(* CODESYS project TestSuite_V1.1.3.library
   Author: Simmel Florian
   Version: 1.1.3
   Title: Tc3_PlcTestSuite
   DefaultNamespace: Tc3_PlcTestSuite
   Placeholder: Tc3_PlcTestSuite
   Company: Simmel

Project tree, tasks and I/O mapping:
  libraries: Tc2_EtherCAT, * (Beckhoff Automation GmbH); Tc2_Standard, * (Beckhoff Automation GmbH); Tc2_System, * (Beckhoff Automation GmbH); Tc2_Utilities, * (Beckhoff Automation GmbH); Tc3_EventLogger, * (Beckhoff Automation GmbH); Tc3_JsonXml, * (Beckhoff Automation GmbH)
  Functions/
    function block AdsLogger [ST]: FB_Init, LogMessage
    function GetValueString [ST]
    function block JUnitResultFile [ST]: AddTestCaseResult, AddTestSuite, AddTestSuiteStatistics, Cyclic, FB_Init, FindSuiteNode, Initialize, Initialized, Path, SaveResult, SuiteOverflowCount
    function block Stopwatch [ST]: Elapsed, Lap, Running, Start, Stop
  Interfaces/
    interface I_TestOperation: AssertEqual, Duration, ExecuteTest, State, TestId, TestSuiteName
    interface I_TestSuite: Duration, ReRunIndividualTest, ReRunTests, Test
    interface I_UnitTestResultFile: AddTestCaseResult, AddTestSuite, AddTestSuiteStatistics, Cyclic, Initialize, Initialized, Path, SaveResult
  Project Information/
    function F_GetCompany [ST]
    function F_GetTitle [ST]
    function F_GetVersion [ST]
  Structures/
    data type E_TestStatus
    data type ST_TestDefinition
  Version/
    global variables Global_Version
  global variables GlobalTestSuite
  function block Test [ST]: AssertEqual, Duration, ExecuteTest, ReportAssert, ResultFileFunction, State, TestId, TestSuiteName
  function block TestSuite [ST]: Duration, FB_Init, ReRunIndividualTest, ReRunTests, ResultFileFunction, Test, TestOverflowCount, TestSuiteName
  global variables TestSuiteParameter
*)

// Structures/E_TestStatus
{attribute 'qualified_only'}
{attribute 'strict'}
{attribute 'to_string'}
TYPE E_TestStatus : (
		Init := 0,
		Running,
		DoneOk,
		DoneFailed
	);
END_TYPE

// Structures/ST_TestDefinition
TYPE ST_TestDefinition :
	STRUCT
		TestId : T_MaxString;
		Status : E_TestStatus;
	END_STRUCT
END_TYPE

// Version/Global_Version
{attribute 'TcGenerated'}
{attribute 'no-analysis'}
{attribute 'linkalways'}
// This function has been automatically generated from the project information.
VAR_GLOBAL CONSTANT
	{attribute 'const_non_replaced'}
	stLibVersion_Tc3_PlcTestSuite : ST_LibVersion := (iMajor := 1, iMinor := 1, iBuild := 3, iRevision := 0, nFlags := 0, sVersion := '1.1.3');
END_VAR

// GlobalTestSuite
VAR_GLOBAL
	JUnitResultFile   : JUnitResultFile<TestSuiteParameter.MaxTestSuiteCount>(TestSuiteParameter.DefaultPath);
	TestSuite		  : TestSuite<TestSuiteParameter.MaxTestCount>(ResultFile := JUnitResultFile);
	AdsLoggingEnabled : BOOL := FALSE;
END_VAR

// TestSuiteParameter
{attribute 'qualified_only'}
VAR_GLOBAL CONSTANT
	MaxTestCount	  : DINT   := 50;
	MaxTestSuiteCount : DINT   := 10;
	DefaultPath		  : STRING := 'C:\ProgramData\Beckhoff\TwinCAT\3.1\Boot\TEST_Result.xml';
END_VAR

// Functions/AdsLogger
FUNCTION_BLOCK AdsLogger
VAR
    Enabled : REFERENCE TO  BOOL;
END_VAR

//FB_Init is always available implicitly and it is used primarily for initialization.
//The return value is not evaluated. For a specific influence, you can also declare the
//methods explicitly and provide additional code there with the standard initialization
//code. You can evaluate the return value.
METHOD FB_Init: BOOL
VAR_INPUT
    bInitRetains: BOOL; // TRUE: the retain variables are initialized (reset warm / reset cold)
    bInCopyCode: BOOL;  // TRUE: the instance will be copied to the copy code afterward (online change) 
    Enabled : REFERENCE TO BOOL;  
END_VAR
THIS^.Enabled Ref= Enabled;
END_METHOD

METHOD LogMessage
VAR_INPUT
	Message : STRING;
END_VAR
IF THIS^.Enabled THEN
	ADSLOGSTR(ADSLOG_MSGTYPE_HINT, Message, '');
END_IF
END_METHOD

END_FUNCTION_BLOCK

// Functions/GetValueString
FUNCTION GetValueString : STRING
VAR_INPUT
	Symbol : ANY;
END_VAR

VAR
	ubuff  : ULINT;
	sibuff : SINT;
	ibuff  : INT;
	dibuff : DINT;
	libuff : LINT;
	rbuff  : REAL;
    lrbuff : LREAL;
	sbuff  : STRING(255);
	wsbuff : WSTRING(255);
	x	   : INT; // loop var for STRING and WSTRING
END_VAR

GetValueString := '';
CASE Symbol.TypeClass OF
	__SYSTEM.TYPE_CLASS.TYPE_BOOL:
		memcpy(ADR(ubuff), Symbol.pValue, TO_UDINT(Symbol.diSize));
		GetValueString := TO_STRING(TO_BOOL(TO_LREAL(ubuff)));

	__SYSTEM.TYPE_CLASS.TYPE_BYTE, __SYSTEM.TYPE_CLASS.TYPE_USINT, __SYSTEM.TYPE_CLASS.TYPE_WORD, __SYSTEM.TYPE_CLASS.TYPE_UINT, __SYSTEM.TYPE_CLASS.TYPE_DWORD, __SYSTEM.TYPE_CLASS.TYPE_UDINT, __SYSTEM.TYPE_CLASS.TYPE_LWORD, __SYSTEM.TYPE_CLASS.TYPE_ULINT:
		memcpy(ADR(ubuff), Symbol.pValue, TO_UDINT(Symbol.diSize));
		GetValueString := LREAL_TO_FMTSTR(TO_LREAL(ubuff), 0, FALSE);

	__SYSTEM.TYPE_CLASS.TYPE_SINT:
		memcpy(ADR(sibuff), Symbol.pValue, TO_UDINT(Symbol.diSize));
		GetValueString := LREAL_TO_FMTSTR(TO_LREAL(sibuff), 0, FALSE);

	__SYSTEM.TYPE_CLASS.TYPE_INT:
		memcpy(ADR(ibuff), Symbol.pValue, TO_UDINT(Symbol.diSize));
		GetValueString := LREAL_TO_FMTSTR(TO_LREAL(ibuff), 0, FALSE);

	__SYSTEM.TYPE_CLASS.TYPE_DINT:
		memcpy(ADR(dibuff), Symbol.pValue, TO_UDINT(Symbol.diSize));
		GetValueString := LREAL_TO_FMTSTR(TO_LREAL(dibuff), 0, FALSE);

	__SYSTEM.TYPE_CLASS.TYPE_LINT:
		memcpy(ADR(libuff), Symbol.pValue, TO_UDINT(Symbol.diSize));
		GetValueString := LREAL_TO_FMTSTR(TO_LREAL(libuff), 0, FALSE);

	__SYSTEM.TYPE_CLASS.TYPE_REAL, __SYSTEM.TYPE_CLASS.TYPE_LREAL:
		IF Symbol.TypeClass = __SYSTEM.TYPE_CLASS.TYPE_REAL THEN
			memcpy(ADR(rbuff), Symbol.pValue, TO_UDINT(Symbol.diSize));
			GetValueString := LREAL_TO_FMTSTR(TO_LREAL(rbuff), 5, TRUE);
		ELSIF Symbol.TypeClass = __SYSTEM.TYPE_CLASS.TYPE_LREAL THEN
			memcpy(ADR(lrbuff), Symbol.pValue, TO_UDINT(Symbol.diSize));
			GetValueString := LREAL_TO_FMTSTR(TO_LREAL(lrbuff), 5, TRUE);
		END_IF

	__SYSTEM.TYPE_CLASS.TYPE_STRING, __SYSTEM.TYPE_CLASS.TYPE_WSTRING:
		IF Symbol.TypeClass = __SYSTEM.TYPE_CLASS.TYPE_STRING THEN
			MEMCPY(ADR(sbuff), Symbol.pValue, MIN(SIZEOF(sbuff), TO_UDINT(Symbol.diSize)));
		ELSIF Symbol.TypeClass = __SYSTEM.TYPE_CLASS.TYPE_WSTRING THEN
			MEMCPY(ADR(wsbuff), Symbol.pValue, MIN(SIZEOF(wsbuff), TO_UDINT(Symbol.diSize)));
			WSTRING_TO_STRING2(ADR(sbuff), ADR(wsbuff), SIZEOF(sbuff));
		END_IF

		GetValueString := sbuff;
END_CASE

END_FUNCTION

// Functions/JUnitResultFile
FUNCTION_BLOCK JUnitResultFile
VAR_GENERIC CONSTANT
	_MaxTestSuiteCount : DINT := 10;
END_VAR IMPLEMENTS I_UnitTestResultFile
VAR
	_Initialized, Write										   : BOOL;
	XmlDomParser											   : FB_XmlDomParser;
	RootNode, TestSuitesNode, TestSuite, TestCase, TestCaseSub : SXmlNode;
	_Path													   : STRING;
	SuiteNames												   : ARRAY[0.._MaxTestSuiteCount] OF STRING;
	SuiteNodes												   : ARRAY[0.._MaxTestSuiteCount] OF SXmlNode;
	SuiteCount												   : DINT;
	DoneMessage												   : FB_TcMessage;
	Source													   : FB_TcSourceInfo;
	_SuiteOverflowCount										   : UDINT;
END_VAR

METHOD AddTestCaseResult
VAR_INPUT
	TestClassName	: STRING;
	TestName		: STRING;
	Duration		: LREAL;
	FailtureMessage : STRING := '';
	FailtureType	: STRING := '';
	FailtureNote	: STRING := '';
END_VAR
VAR
	SuiteNode : SXmlNode;
END_VAR
IF NOT Initialized THEN
	RETURN;
END_IF

SuiteNode := FindSuiteNode(TestClassName);
IF SuiteNode = 0 THEN
	RETURN;
END_IF

TestCase := XmlDomParser.AppendChild(SuiteNode,
									 'testcase',
									 '',
									 FALSE);

XmlDomParser.AppendAttribute(TestCase, 'classname', TestClassName);
XmlDomParser.AppendAttribute(TestCase, 'name', TestName);
XmlDomParser.AppendAttributeAsDouble(TestCase, 'time', Duration);
IF FailtureType <> '' THEN
	TestCaseSub := XmlDomParser.AppendChild(TestCase,
											'failure',
											FailtureNote,
											FALSE);

	XmlDomParser.AppendAttribute(TestCaseSub, 'message', FailtureMessage);
	XmlDomParser.AppendAttribute(TestCaseSub, 'type', FailtureType);
END_IF
END_METHOD

METHOD AddTestSuite
VAR_INPUT
	Name : STRING;
END_VAR
VAR
	ResultString : T_MaxString;
END_VAR
IF NOT Initialized THEN
	RETURN;
END_IF

// Reuse the existing node if this suite name was already added (shared result file across multiple TestSuite instances)
TestSuite := FindSuiteNode(Name);
IF TestSuite <> 0 THEN
	RETURN;
END_IF

TestSuite := XmlDomParser.AppendChild(TestSuitesNode,
									  'testsuite',
									  '',
									  FALSE);

XmlDomParser.AppendAttribute(TestSuite, 'name', name);

IF SuiteCount <= _MaxTestSuiteCount THEN
	SuiteNames[SuiteCount] := Name;
	SuiteNodes[SuiteCount] := TestSuite;
	SuiteCount			   := SuiteCount + 1;
ELSE
	_SuiteOverflowCount := _SuiteOverflowCount + 1;

	Source.sName := Name;
	DoneMessage.Create(eventClass	:= TC_EVENT_CLASSES.TestEvents,
					   nEventId		:= 1,
					   eSeverity	:= TcEventSeverity.Error,
					   ipSourceInfo := Source);

	ResultString := CONCAT('TestSuite not added, max TestSuites exeeded - ', TO_STRING(_MaxTestSuiteCount));
	DoneMessage.ipArguments.AddString(ResultString);
	DoneMessage.Send(0);
	Source.Clear();
	DoneMessage.Release();
END_IF
END_METHOD

METHOD AddTestSuiteStatistics
VAR_INPUT
	Name	  : STRING;
	Tests	  : UDINT;
	Failtures : UDINT := 0;
	Errors	  : UDINT := 0;
	Skipped	  : UDINT := 0;
	Duration  : LREAL;
END_VAR
VAR
	SuiteNode : SXmlNode;
END_VAR
IF NOT Initialized THEN
	RETURN;
END_IF

SuiteNode := FindSuiteNode(Name);
IF SuiteNode = 0 THEN
	RETURN;
END_IF

XmlDomParser.AppendAttributeAsUint(SuiteNode, 'tests', Tests);
XmlDomParser.AppendAttributeAsUint(SuiteNode, 'failtures', Failtures);
XmlDomParser.AppendAttributeAsUint(SuiteNode, 'errors', Errors);
XmlDomParser.AppendAttributeAsUint(SuiteNode, 'skipped', Skipped);
XmlDomParser.AppendAttributeAsDouble(SuiteNode, 'time', Duration);
END_METHOD

METHOD Cyclic
XmlDomParser.SaveDocumentToFile(_Path, Write);
END_METHOD

//FB_Init is always available implicitly and it is used primarily for initialization.

//The return value is not evaluated. For a specific influence, you can also declare the

//methods explicitly and provide additional code there with the standard initialization

//code. You can evaluate the return value.
METHOD FB_Init : BOOL
VAR_INPUT
	bInitRetains : BOOL; // TRUE: the retain variables are initialized (reset warm / reset cold)
	bInCopyCode	 : BOOL; // TRUE: the instance will be copied to the copy code afterward (online change)
	Path		 : STRING;
END_VAR
_Path := Path;
END_METHOD

METHOD PRIVATE FindSuiteNode : SXmlNode
VAR_INPUT
	Name : STRING;
END_VAR
VAR
	i : DINT;
END_VAR
FindSuiteNode := 0;

FOR i := 0 TO SuiteCount - 1 DO
	IF SuiteNames[i] = Name THEN
		FindSuiteNode := SuiteNodes[i];
		RETURN;
	END_IF
END_FOR
END_METHOD

METHOD Initialize
VAR_INPUT
	ReInitialize : BOOL := FALSE;
END_VAR
IF Initialized AND NOT ReInitialize THEN
	RETURN;
END_IF

XmlDomParser.NewDocument();
RootNode	   := XmlDomParser.GetDocumentNode();
TestSuitesNode := XmlDomParser.AppendChild(RootNode,
										   'testsuites',
										   '',
										   FALSE);

SuiteCount	 := 0;
_Initialized := TRUE;
END_METHOD

{attribute 'monitoring' := 'call'}
PROPERTY Initialized : BOOL
GET
Initialized := _Initialized;
END_GET
END_PROPERTY

{attribute 'monitoring' := 'call'}
PROPERTY Path : STRING
SET
_Path := Path;
END_SET
END_PROPERTY

METHOD SaveResult
IF NOT Initialized THEN
	RETURN;
END_IF

Write := TRUE;
END_METHOD

{attribute 'monitoring' := 'call'}
PROPERTY SuiteOverflowCount : UDINT
GET
SuiteOverflowCount := _SuiteOverflowCount;
END_GET
END_PROPERTY

END_FUNCTION_BLOCK

// Interfaces/I_UnitTestResultFile
INTERFACE I_UnitTestResultFile EXTENDS __SYSTEM.IQueryInterface

METHOD AddTestCaseResult
VAR_INPUT
	TestClassName	: STRING;
	TestName		: STRING;
	Duration		: LREAL;
	FailtureMessage : STRING := '';
	FailtureType	: STRING := '';
	FailtureNote	: STRING := '';
END_VAR
END_METHOD

METHOD AddTestSuite
VAR_INPUT
	Name	  : STRING;
END_VAR
END_METHOD

METHOD AddTestSuiteStatistics
VAR_INPUT
	Name	  : STRING;
	Tests	  : UDINT;
	Failtures : UDINT := 0;
	Errors	  : UDINT := 0;
	Skipped	  : UDINT := 0;
	Duration  : LREAL;
END_VAR
END_METHOD

METHOD Cyclic
VAR_INPUT
END_VAR
END_METHOD

METHOD Initialize
VAR_INPUT
	ReInitialize : BOOL := FALSE;
END_VAR
END_METHOD

{attribute 'monitoring' := 'call'}
PROPERTY Initialized : BOOL
GET
END_GET
END_PROPERTY

{attribute 'monitoring' := 'call'}
PROPERTY Path : STRING
SET
END_SET
END_PROPERTY

METHOD SaveResult
VAR_INPUT
END_VAR
END_METHOD

END_INTERFACE

// TestSuite
FUNCTION_BLOCK TestSuite
VAR_GENERIC CONSTANT
	_MaxTestCount : DINT := 10;
END_VAR IMPLEMENTS I_TestSuite
VAR
	_TestSuiteName	  : STRING;
	TestCollection	  : ARRAY[0.._MaxTestCount] OF Test;
	NoAction		  : Test := (TestId := 'No Action', State := E_TestStatus.DoneOk);
	ActiveTest		  : DINT;
	DoneMessage		  : FB_TcMessage;
	Source			  : FB_TcSourceInfo;
	TotalTestCount	  : UDINT := 0;
	TotalOkTestCount  : UDINT := 0;
	TotalNokTestCount : UDINT := 0;
	Complete		  : BOOL;
	ResultFile		  : I_UnitTestResultFile;
	_ResultFileAdded  : BOOL;
	CurrentCycle	  : UDINT;
	Stopwatch		  : Stopwatch;
	_TestOverflowCount : UDINT;
END_VAR

{attribute 'monitoring' := 'call'}
PROPERTY Duration : LREAL
GET
Duration := Stopwatch.Elapsed;
END_GET
END_PROPERTY

//FB_Init is always available implicitly and it is used primarily for initialization.

//The return value is not evaluated. For a specific influence, you can also declare the

//methods explicitly and provide additional code there with the standard initialization

//code. You can evaluate the return value.
METHOD FB_Init : BOOL
VAR_INPUT
	bInitRetains : BOOL; // TRUE: the retain variables are initialized (reset warm / reset cold)
	bInCopyCode	 : BOOL; // TRUE: the instance will be copied to the copy code afterward (online change)
	ResultFile	 : I_UnitTestResultFile;
END_VAR
IF ResultFile <> 0 THEN
	THIS^.ResultFile := ResultFile;
END_IF
END_METHOD

{attribute 'TcRpcEnable':='1'}
METHOD ReRunIndividualTest
VAR_INPUT
	TestId : T_MaxString;
END_VAR

VAR
	i : DINT;
END_VAR
FOR i := 0 TO _MaxTestCount DO
	IF TestCollection[i].TestId = TestId THEN
		TestCollection[i].State := E_TestStatus.Init;
		ActiveTest := i;
		Complete := FALSE;
		EXIT;
	END_IF
END_FOR
END_METHOD

{attribute 'TcRpcEnable':='1'}
METHOD ReRunTests
VAR
	i : DINT;
END_VAR
FOR i := 0 TO TestSuiteParameter.MaxTestCount DO
	TestCollection[i].State := E_TestStatus.Init;
	ActiveTest				:= 0;
	Complete				:= FALSE;
	ResultFile.Initialize();
	Stopwatch.Start();
	ResultFile.AddTestSuite(Name := _TestSuiteName);
END_FOR
END_METHOD

PROPERTY ResultFileFunction : I_UnitTestResultFile
SET
ResultFile := ResultFileFunction;
END_SET
END_PROPERTY

METHOD Test : I_TestOperation
VAR_INPUT
	TestId : T_MaxString;
END_VAR

VAR
	ResultString : T_MaxString;
	i			 : DINT;
END_VAR
IF _TestSuiteName = '' THEN
	_TestSuiteName := __POUNAME();
END_IF

IF NOT _ResultFileAdded THEN
	_ResultFileAdded := TRUE;
	ResultFile.Initialize();
	Stopwatch.Start();
	ResultFile.AddTestSuite(Name := _TestSuiteName);
END_IF

IF TwinCAT_SystemInfoVarList._TaskInfo[GETCURTASKINDEXEX()].CycleCount <> CurrentCycle THEN
	CurrentCycle := TwinCAT_SystemInfoVarList._TaskInfo[GETCURTASKINDEXEX()].CycleCount;
	ResultFile.Cyclic();
END_IF

IF NOT Complete THEN
	FOR i := 0 TO _MaxTestCount DO
		TestCollection[i].TestSuiteName		 := _TestSuiteName;
		TestCollection[i].ResultFileFunction := ResultFile;
		// Detect first running test
		IF TestCollection[i].State = E_TestStatus.Running THEN
			ActiveTest := i;
		END_IF

		IF TestCollection[ActiveTest].State >= E_TestStatus.DoneOk THEN
			ActiveTest := 0;
		END_IF

		// Get existing Test
		IF (TestCollection[i].TestId = TestId) THEN
			IF (ActiveTest = i) OR (ActiveTest = 0) THEN
				Test := TestCollection[i];
			ELSE
				Test := NoAction;
			END_IF

			EXIT;
		END_IF

		// Add Test
		IF TestCollection[i].TestId = '' THEN
			TestCollection[i].TestId := TestId;
			Test					 := NoAction;
			EXIT;
		END_IF

		// Out of tests
		IF i = _MaxTestCount THEN
			Test			   := NoAction;
			_TestOverflowCount := _TestOverflowCount + 1;
			Source.sName	   := _TestSuiteName;
			DoneMessage.Create(eventClass	:= TC_EVENT_CLASSES.TestEvents,
							   nEventId		:= 1,
							   eSeverity	:= TcEventSeverity.Error,
							   ipSourceInfo := Source);

			ResultString := CONCAT('Test not added, max Tests exeeded - ', TO_STRING(_MaxTestCount));
			DoneMessage.ipArguments.AddString(ResultString);
			DoneMessage.Send(0);
			Source.Clear();
			DoneMessage.Release();
			Complete := TRUE;
		END_IF
	END_FOR

	// Run Statistic
	TotalTestCount	  := 0;
	TotalOkTestCount  := 0;
	TotalNokTestCount := 0;
	FOR i := 0 TO _MaxTestCount DO
		IF TestCollection[i].TestId <> '' THEN
			TotalTestCount := TotalTestCount + 1;
			IF TestCollection[i].State = E_TestStatus.DoneOk THEN
				TotalOkTestCount := TotalOkTestCount + 1;
			END_IF

			IF TestCollection[i].State = E_TestStatus.DoneFailed THEN
				TotalNokTestCount := TotalNokTestCount + 1;
			END_IF
		END_IF
	END_FOR

	// Tests finished
	IF (TotalTestCount = (TotalOkTestCount + TotalNokTestCount)) AND NOT Complete THEN
		Source.sName := _TestSuiteName;
		DoneMessage.Create(eventClass	:= TC_EVENT_CLASSES.TestEvents,
						   nEventId		:= 1,
						   eSeverity	:= TcEventSeverity.Error,
						   ipSourceInfo := Source);

		ResultString := CONCAT('Completed - ', CONCAT('Total Tests - ', TO_STRING(TotalTestCount)));
		ResultString := CONCAT(ResultString, CONCAT(', OK Tests - ', TO_STRING(TotalOkTestCount)));
		ResultString := CONCAT(ResultString, CONCAT(', Failed Tests - ', TO_STRING(TotalNokTestCount)));
		DoneMessage.ipArguments.AddString(ResultString);
		DoneMessage.Send(0);
		Source.Clear();
		DoneMessage.Release();

		//
		Stopwatch.Stop();
		ResultFile.AddTestSuiteStatistics(Name := _TestSuiteName, Tests := TotalTestCount, Failtures := TotalNokTestCount, Duration := Stopwatch.Elapsed);
		ResultFile.SaveResult();

		//
		Complete := TRUE;
	END_IF
ELSE
	Test := NoAction;
END_IF
END_METHOD

{attribute 'monitoring' := 'call'}
PROPERTY TestOverflowCount : UDINT
GET
TestOverflowCount := _TestOverflowCount;
END_GET
END_PROPERTY

{attribute 'monitoring' := 'call'}
PROPERTY TestSuiteName : STRING
SET
_TestSuiteName := TestSuiteName;
END_SET
END_PROPERTY

END_FUNCTION_BLOCK

// Interfaces/I_TestSuite
INTERFACE I_TestSuite EXTENDS __SYSTEM.IQueryInterface

{attribute 'monitoring' := 'call'}
PROPERTY Duration : LREAL
GET
END_GET
END_PROPERTY

METHOD ReRunIndividualTest
VAR_INPUT
	TestId : T_MaxString;
END_VAR
END_METHOD

METHOD ReRunTests
VAR_INPUT
END_VAR
END_METHOD

METHOD Test : I_TestOperation
VAR_INPUT
	TestId : T_MaxString;
END_VAR
END_METHOD

END_INTERFACE

// Test
FUNCTION_BLOCK Test IMPLEMENTS I_TestOperation
VAR
	_TestSuiteName : STRING;
	_TestId		   : T_MaxString;
	_State		   : E_TestStatus;
	TestMessage	   : FB_TcMessage;
	Source		   : FB_TcSourceInfo;
	Stopwatch	   : Stopwatch;
	ResultFile	   : I_UnitTestResultFile;
	AdsLogger	   : AdsLogger(GlobalTestSuite.AdsLoggingEnabled);
END_VAR

METHOD AssertEqual
VAR_INPUT
	Expected : ANY;
	Actual	 : ANY;
	Epsilon	 : LREAL := 0.000001;
END_VAR

VAR
	nCount		   : DINT;
	StringExpected : T_MaxString;
	StringActual   : T_MaxString;
	LrealExpected  : LREAL;
	LrealActual	   : LREAL;
	RealExpected   : REAL;
	RealActual	   : REAL;
END_VAR
Stopwatch.Stop();
IF Expected.typeclass <> Actual.typeclass THEN
	State := E_TestStatus.DoneFailed;
	ReportAssert('Type missmatch!');
	RETURN;
END_IF

IF Expected.diSize <> Actual.diSize THEN
	State := E_TestStatus.DoneFailed;
	ReportAssert('Type size missmatch!');
	RETURN;
END_IF

// String
IF Expected.TypeClass = __SYSTEM.TYPE_CLASS.TYPE_ANYSTRING OR Expected.TypeClass = __SYSTEM.TYPE_CLASS.TYPE_STRING OR Expected.TypeClass = __SYSTEM.TYPE_CLASS.TYPE_WSTRING OR Expected.TypeClass = __SYSTEM.TYPE_CLASS.TYPE_XSTRING THEN
	MEMCPY(destAddr := ADR(StringExpected), srcAddr := Expected.pValue, n := DINT_TO_UDINT(Expected.diSize));
	MEMCPY(destAddr := ADR(StringActual), srcAddr := Actual.pValue, n := DINT_TO_UDINT(Actual.diSize));
	IF StringExpected <> StringActual THEN
		State := E_TestStatus.DoneFailed;
		ReportAssert(CONCAT(CONCAT('Expected: ', GetValueString(Expected)), CONCAT(' , Actual: ', GetValueString(Actual))));
		RETURN;
	END_IF
ELSIF Expected.TypeClass = __SYSTEM.TYPE_CLASS.TYPE_LREAL THEN
	MEMCPY(destAddr := ADR(LrealExpected), srcAddr := Expected.pValue, n := DINT_TO_UDINT(Expected.diSize));
	MEMCPY(destAddr := ADR(LrealActual), srcAddr := Actual.pValue, n := DINT_TO_UDINT(Actual.diSize));
	IF ((LrealExpected - Epsilon) > LrealActual) OR ((LrealExpected + Epsilon) < LrealActual) THEN
		State := E_TestStatus.DoneFailed;
		ReportAssert(CONCAT(CONCAT('Expected: ', GetValueString(Expected)), CONCAT(' , Actual: ', GetValueString(Actual))));
		RETURN;
	END_IF
ELSIF Expected.TypeClass = __SYSTEM.TYPE_CLASS.TYPE_ANYREAL OR Expected.TypeClass = __SYSTEM.TYPE_CLASS.TYPE_REAL THEN
	MEMCPY(destAddr := ADR(RealExpected), srcAddr := Expected.pValue, n := DINT_TO_UDINT(Expected.diSize));
	MEMCPY(destAddr := ADR(RealActual), srcAddr := Actual.pValue, n := DINT_TO_UDINT(Actual.diSize));
	IF ((RealExpected - Epsilon) > RealActual) OR ((RealExpected + Epsilon) < RealActual) THEN
		State := E_TestStatus.DoneFailed;
		ReportAssert(CONCAT(CONCAT('Expected: ', GetValueString(Expected)), CONCAT(' , Actual: ', GetValueString(Actual))));
		RETURN;
	END_IF
ELSE
	// Byte comparison
	FOR nCount := 0 TO Actual.diSize - 1 DO
		IF Expected.pvalue[nCount] <> Actual.pvalue[nCount] THEN
			State := E_TestStatus.DoneFailed;
			ReportAssert(CONCAT(CONCAT('Expected: ', GetValueString(Expected)), CONCAT(' , Actual: ', GetValueString(Actual))));
			RETURN;
		END_IF
	END_FOR
END_IF

IF ResultFile <> 0 THEN
	ResultFile.AddTestCaseResult(_TestSuiteName, TestId, Stopwatch.Elapsed);
END_IF

AdsLogger.LogMessage(Concat('Test Executed: ', TestId));
State := E_TestStatus.DoneOk;
END_METHOD

{attribute 'monitoring' := 'call'}
PROPERTY Duration : LREAL
GET
Duration := Stopwatch.Elapsed;
END_GET
END_PROPERTY

METHOD ExecuteTest : BOOL
VAR_INPUT
END_VAR
IF State = E_TestStatus.Init THEN
	Stopwatch.Start();
	State := E_TestStatus.Running;
END_IF

ExecuteTest := State = E_TestStatus.Running;
END_METHOD

METHOD PRIVATE ReportAssert
VAR_INPUT
	Reason : STRING := '';
END_VAR

VAR
	ResultString : T_MaxString;
END_VAR
Source.sName := _TestSuiteName;
TestMessage.Create(eventClass	:= TC_EVENT_CLASSES.TestEvents,
				   nEventId		:= 1,
				   eSeverity	:= TcEventSeverity.Error,
				   ipSourceInfo := Source);

ResultString := CONCAT('Test failed - ', TestId);
ResultString := CONCAT(ResultString, '! ');
ResultString := CONCAT(ResultString, Reason);
TestMessage.ipArguments.AddString(ResultString);
TestMessage.Send(0);
Source.Clear();
TestMessage.Release();
AdsLogger.LogMessage(Concat('Test Executed: ', TestId));
IF ResultFile <> 0 THEN
	ResultFile.AddTestCaseResult(_TestSuiteName,
								 TestId,
								 Stopwatch.Elapsed,
								 'Test failed!',
								 'AssertionError',
								 Reason);
END_IF
END_METHOD

PROPERTY ResultFileFunction : I_UnitTestResultFile
SET
ResultFile := ResultFileFunction;
END_SET
END_PROPERTY

{attribute 'monitoring' := 'call'}
PROPERTY State :  E_TestStatus
GET
State := _State;
END_GET
SET
_State := State;
END_SET
END_PROPERTY

{attribute 'monitoring' := 'call'}
PROPERTY TestId : T_MaxString
GET
TestId := _TestId;
END_GET
SET
_TestId := TestId;
END_SET
END_PROPERTY

{attribute 'monitoring' := 'call'}
PROPERTY TestSuiteName : STRING
SET
_TestSuiteName := TestSuiteName;
END_SET
END_PROPERTY

END_FUNCTION_BLOCK

// Interfaces/I_TestOperation
INTERFACE I_TestOperation EXTENDS __SYSTEM.IQueryInterface

METHOD AssertEqual
VAR_INPUT
	Expected : ANY;
	Actual	 : ANY;
	Epsilon	 : LREAL := 0.000001;
END_VAR
END_METHOD

{attribute 'monitoring' := 'call'}
PROPERTY Duration : LREAL
GET
END_GET
END_PROPERTY

METHOD ExecuteTest : BOOL
VAR_INPUT
END_VAR
END_METHOD

{attribute 'monitoring' := 'call'}
PROPERTY State : E_TestStatus
GET
END_GET
SET
END_SET
END_PROPERTY

{attribute 'monitoring' := 'call'}
PROPERTY TestId : T_MaxString
GET
END_GET
SET
END_SET
END_PROPERTY

{attribute 'monitoring' := 'call'}
PROPERTY TestSuiteName : String
SET
END_SET
END_PROPERTY

END_INTERFACE

// Functions/Stopwatch
FUNCTION_BLOCK Stopwatch
VAR
	StartTime			: T_DCTIME64;
	EndTime				: T_DCTIME64;
	PreviousLapEndTime	: T_DCTIME64;
	PreviousElapsedTime : LREAL;
	_Running			: BOOL;
END_VAR

VAR CONSTANT
	OneNanosecond : LREAL := 1.0E-9;
END_VAR

{attribute 'monitoring' := 'call'}
PROPERTY Elapsed : LREAL
GET
IF _Running THEN
	Elapsed := TO_LREAL(F_GetCurDcTickTime64() - StartTime) * OneNanosecond;
ELSE
	Elapsed := PreviousElapsedTime;
END_IF
END_GET
END_PROPERTY

METHOD Lap : LREAL;
VAR
	LapEndTime	: T_DCTIME64;
	LapDuration : LREAL;
END_VAR
IF _Running THEN
	LapEndTime		   := F_GetActualDcTime64();
	LapDuration		   := TO_LREAL(LapEndTime - PreviousLapEndTime) * OneNanosecond;
	PreviousLapEndTime := LapEndTime;
	Lap				   := LapDuration;
END_IF
END_METHOD

{attribute 'monitoring' := 'call'}
PROPERTY Running : BOOL
GET
Running := _Running;
END_GET
END_PROPERTY

METHOD Start
StartTime			:= F_GetActualDcTime64();
PreviousLapEndTime	:= StartTime;
_Running			:= TRUE;
PreviousElapsedTime := 0.0;
PreviousElapsedTime := 0;
END_METHOD

METHOD Stop : LREAL
IF _Running THEN
	EndTime				:= F_GetActualDcTime64();
	_Running			:= FALSE;
	PreviousElapsedTime := TO_LREAL(EndTime - StartTime) * OneNanosecond;
	Stop				:= PreviousElapsedTime;
ELSE
	Stop := 0.0;
END_IF
END_METHOD

END_FUNCTION_BLOCK

// Project Information/F_GetCompany
// This function has been automatically generated from the project information.
{attribute 'signature_flag' := '1073741824'}
{attribute 'TcGenerated'}
{attribute 'no-analysis'}
FUNCTION F_GetCompany : WSTRING
VAR_INPUT
	
END_VAR

F_GetCompany := "Simmel";

END_FUNCTION

// Project Information/F_GetTitle
// This function has been automatically generated from the project information.
{attribute 'signature_flag' := '1073741824'}
{attribute 'TcGenerated'}
{attribute 'no-analysis'}
FUNCTION F_GetTitle : WSTRING
VAR_INPUT
	
END_VAR

F_GetTitle := "Tc3_PlcTestSuite";

END_FUNCTION

// Project Information/F_GetVersion
// This function has been automatically generated from the project information.
{attribute 'signature_flag' := '1073741824'}
{attribute 'TcGenerated'}
{attribute 'no-analysis'}
FUNCTION F_GetVersion : ST_LibVersion
VAR_INPUT
	
END_VAR

F_GetVersion.iMajor := 1;
F_GetVersion.iMinor := 1;
F_GetVersion.iBuild := 3;
F_GetVersion.iRevision := 0;
F_GetVersion.sVersion := '1.1.3';
F_GetVersion.nFlags := 0;

END_FUNCTION
